{attribute 'qualified_only'}
VAR_GLOBAL
	Axis: AXIS_REF;
END_VAR

(* stored: Version 1.1.0.1, ProductVersion 3.1.4024.12
   GVL GVL: Id {58e4746b-de9a-4f4e-9d82-0c44aa0be39b} *)
